Universal Robots PolyScope program: 3_pickup_glass_to_hover.urp

Program 3_pickup_glass_to_hover (installation=default directory=/programs/washer_rahman createdIn=5.9.5.1031259 lastSavedIn=5.9.5.1031259 robotSerialNumber=20215500597)
Calibrated DH parameters: a=[0.000193, -0.066673, -0.391568, -0.000012, 0.00005, 0]; d=[0.162643, -472.05677, 465.132521, 7.058239, 0.099746, 0.099582]; alpha=[1.571116, 0.00089, 0.003862, 1.569269, -1.569248, 0]; deltaTheta=[0, -1.413394, 7.628392, 0.068187, 0, -0.000001]
Robot Program (runOnlyOnce=true)
  SuppressedNode
    MoveL speed 250 mm/s, acceleration 1200 mm/s^2 (useActiveTCP=true) feature=Base
      MoveDirectionNode (selectedDirection=ZMinus)
        Until DISTANCE (allowActions=false deceleration=3 distanceNodeType=STOP) Distance=0.07; motionParameters(blendRadius=0)
  SuppressedNode
    URCap Gripper (Robotiq_Grippers, Robotiq Inc.) dataModel(position=32.94117647058823, force=100.0, speed=100.0, positionInDouble=32.94117647058823, forceInDouble=100.0, speedInDouble=100.0, slaveIds=[9], blocking=true)
  MoveL speed 250 mm/s, acceleration 1200 mm/s^2 (useActiveTCP=true) feature=Base
    Waypoint Waypoint_2: TCP in base x=-566.064 y=-176.539 z=307.289 mm, rx=-1.2228 ry=-1.3732 rz=1.1429 rad; joints [5.32, -79.631, 138.52, -231.6, -92.319, -3.015] deg; TCP offset x=0 y=0 z=191.5 mm, rx=0 ry=0 rz=0 rad
    MoveDirectionNode (selectedDirection=ZPlus)
      Until DISTANCE (allowActions=false deceleration=3 distanceNodeType=STOP) Distance=0.15; motionParameters(blendRadius=0)
    MoveJ speed 60 deg/s, acceleration 80 deg/s^2 (useActiveTCP=true) feature=Base
      Waypoint Waypoint_1: TCP in base x=-570.315 y=-142.132 z=406.221 mm, rx=-1.2552 ry=-1.3745 rz=1.0423 rad; joints [2.423, -96.242, 131.84, -205.844, -93.339, -5.251] deg
